{attribute 'qualified_only'}
TYPE E_PackMLState :
(
    Undefined    := 0,
    Clearing     := 1,
    Stopped      := 2,
    Starting     := 3,
    Idle         := 4,
    Suspended    := 5,
    Execute      := 6,
    Stopping     := 7,
    Aborting     := 8,
    Aborted      := 9,
    Holding      := 10,
    Held         := 11,
    Unholding    := 12,
    Suspending   := 13,
    Unsuspending := 14,
    Resetting    := 15,
    Completing   := 16,
    Complete     := 17
);
END_TYPE

(* stored: Version 1.1.0.1, ProductVersion 3.1.4024.16
   DUT DUT: Id {64b82f68-cdcb-4063-b058-c8995e1bf43a} *)
